// TIA Portal V20 export
// export: Created 2026-04-11T06:02:30.4295943Z, ExportSetting WithDefaults, DisplayName Totally Integrated Automation Portal, DisplayVersion V20, DisplayName TIA Portal Openness, DisplayVersion V20, DisplayName TIA Portal Version Control Interface, DisplayVersion V20, DisplayName STEP 7 Professional, DisplayVersion V20, DisplayName STEP 7 Safety, DisplayVersion V20, DisplayName WinCC Basic/Comfort/Advanced, DisplayVersion V20, DisplayName WinCC Unified, DisplayVersion V20
TYPE "udtHMI_Interlock"
// stored: IsFailsafeCompliant false
   STRUCT
      abInterlocks { ExternalWritable := 'False'} : Array[1..16] of Bool;   // Interlock statuses
      asInterlockNames { S7_SetPoint := 'True'} : Array[1..16] of String[20];   // Interlock names
      bInterlockOk { ExternalWritable := 'False'} : Bool;   // System Interlock is ok
   END_STRUCT;
END_TYPE
